// TIA Portal V18 export
// export: Created 2026-01-09T11:31:59.1599662Z, ExportSetting WithDefaults, DisplayName Totally Integrated Automation Portal, DisplayVersion V18 Update 5, DisplayName TIA Portal Openness, DisplayVersion V18 Update 5, DisplayName TIA Portal Teamcenter Gateway, DisplayVersion V18, DisplayName TIA Portal Version Control Interface, DisplayVersion V18, DisplayName SINAMICS Startdrive Advanced, DisplayVersion V18 SP2 Update 1, DisplayName SINAMICS Startdrive G110M, G120, G120C, G120D, G120P, G115D, DisplayVersion V18 SP2 Update 1, DisplayName SINAMICS Startdrive G130, G150, S120, S150, SINAMICS MV, S210, G220, S200, DisplayVersion V18 SP2 Update 1, DisplayName STEP 7 Professional, DisplayVersion V18 Update 5, DisplayName STEP 7 Safety, DisplayVersion V18, DisplayName WinCC Professional, DisplayVersion V18 Update 5
TagTable "WarningWord"
  GlobalWarning_01 : Word  (%DB1068.DBW0, CPU S71500-2PN_TP700, 100 ms)
  GlobalWarning_02 : Word  (%DB1068.DBW2, CPU S71500-2PN_TP700, 100 ms)
  GlobalWarning_03 : Word  (%DB1068.DBW4, CPU S71500-2PN_TP700, 100 ms)
  GlobalWarning_04 : Word  (%DB1068.DBW6, CPU S71500-2PN_TP700, 100 ms)
  GlobalWarning_05 : Word  (%DB1068.DBW8, CPU S71500-2PN_TP700, 100 ms)
  GlobalWarning_06 : Word  (%DB1068.DBW10, CPU S71500-2PN_TP700, 100 ms)
  GlobalWarning_07 : Word  (%DB1068.DBW12, CPU S71500-2PN_TP700, 100 ms)
  GlobalWarning_08 : Word  (%DB1068.DBW14, CPU S71500-2PN_TP700, 100 ms)
  GlobalWarning_09 : Word  (%DB1068.DBW16, CPU S71500-2PN_TP700, 100 ms)
  GlobalWarning_10 : Word  (%DB1068.DBW18, CPU S71500-2PN_TP700, 100 ms)
  IndexTableWarning_01 : Word  (%DB1068.DBW20, CPU S71500-2PN_TP700, 100 ms)
  IndexTableWarning_02 : Word  (%DB1068.DBW22, CPU S71500-2PN_TP700, 100 ms)
  ServoWarning_01 : Word  (%DB1068.DBW24, CPU S71500-2PN_TP700, 100 ms)
  ServoWarning_02 : Word  (%DB1068.DBW26, CPU S71500-2PN_TP700, 100 ms)
  ServePressWarning_01 : Word  (%DB1068.DBW28, CPU S71500-2PN_TP700, 100 ms)
  ServePressWarning_02 : Word  (%DB1068.DBW30, CPU S71500-2PN_TP700, 100 ms)
  3AxisInterpolationWarning_01 : Word  (%DB1068.DBW32, CPU S71500-2PN_TP700, 100 ms)
  3AxisInterpolationWarning_02 : Word  (%DB1068.DBW34, CPU S71500-2PN_TP700, 100 ms)
  LaserWeldingWarning_01 : Word  (%DB1068.DBW36, CPU S71500-2PN_TP700, 100 ms)
  LaserWeldingWarning_02 : Word  (%DB1068.DBW38, CPU S71500-2PN_TP700, 100 ms)
  LaserMarkingWarning_01 : Word  (%DB1068.DBW40, CPU S71500-2PN_TP700, 100 ms)
  LaserMarkingWarning_02 : Word  (%DB1068.DBW42, CPU S71500-2PN_TP700, 100 ms)
  PrinterWarning_01 : Word  (%DB1068.DBW44, CPU S71500-2PN_TP700, 100 ms)
  PrinterWarning_02 : Word  (%DB1068.DBW46, CPU S71500-2PN_TP700, 100 ms)
  MarkingWarning_01 : Word  (%DB1068.DBW48, CPU S71500-2PN_TP700, 100 ms)
  MarkingWarning_02 : Word  (%DB1068.DBW50, CPU S71500-2PN_TP700, 100 ms)
  LabellingWarning_01 : Word  (%DB1068.DBW52, CPU S71500-2PN_TP700, 100 ms)
  LabellingWarning_02 : Word  (%DB1068.DBW54, CPU S71500-2PN_TP700, 100 ms)
  DispensingWarning_01 : Word  (%DB1068.DBW56, CPU S71500-2PN_TP700, 100 ms)
  DispensingWarning_02 : Word  (%DB1068.DBW58, CPU S71500-2PN_TP700, 100 ms)
  GreasingWarning_01 : Word  (%DB1068.DBW60, CPU S71500-2PN_TP700, 100 ms)
  GreasingWarning_02 : Word  (%DB1068.DBW62, CPU S71500-2PN_TP700, 100 ms)
  HotWindSystemWarning_01 : Word  (%DB1068.DBW64, CPU S71500-2PN_TP700, 100 ms)
  HotWindSystemWarning_02 : Word  (%DB1068.DBW66, CPU S71500-2PN_TP700, 100 ms)
  HighFrequencyHeatingWarning_01 : Word  (%DB1068.DBW68, CPU S71500-2PN_TP700, 100 ms)
  HighFrequencyHeatingWarning_02 : Word  (%DB1068.DBW70, CPU S71500-2PN_TP700, 100 ms)
  DegaussingWarning_01 : Word  (%DB1068.DBW72, CPU S71500-2PN_TP700, 100 ms)
  DegaussingWarning_02 : Word  (%DB1068.DBW74, CPU S71500-2PN_TP700, 100 ms)
  BowlFeederWarning_01 : Word  (%DB1068.DBW76, CPU S71500-2PN_TP700, 100 ms)
  BowlFeederWarning_02 : Word  (%DB1068.DBW78, CPU S71500-2PN_TP700, 100 ms)
  RiveterWarning_01 : Word  (%DB1068.DBW80, CPU S71500-2PN_TP700, 100 ms)
  RiveterWarning_02 : Word  (%DB1068.DBW82, CPU S71500-2PN_TP700, 100 ms)
  HydraulicSystemWarning_01 : Word  (%DB1068.DBW84, CPU S71500-2PN_TP700, 100 ms)
  HydraulicSystemWarning_02 : Word  (%DB1068.DBW86, CPU S71500-2PN_TP700, 100 ms)
  RobotWarning_01 : Word  (%DB1068.DBW88, CPU S71500-2PN_TP700, 100 ms)
  RobotWarning_02 : Word  (%DB1068.DBW90, CPU S71500-2PN_TP700, 100 ms)
  CameraWarning_01 : Word  (%DB1068.DBW92, CPU S71500-2PN_TP700, 100 ms)
  CameraWarning_02 : Word  (%DB1068.DBW94, CPU S71500-2PN_TP700, 100 ms)
  ScannnerWarning_01 : Word  (%DB1068.DBW96, CPU S71500-2PN_TP700, 100 ms)
  ScannnerWarning_02 : Word  (%DB1068.DBW98, CPU S71500-2PN_TP700, 100 ms)
  MeasureSensorWarning_01 : Word  (%DB1068.DBW100, CPU S71500-2PN_TP700, 100 ms)
  MeasureSensorWarning_02 : Word  (%DB1068.DBW102, CPU S71500-2PN_TP700, 100 ms)
  LeakageTesterWarning_01 : Word  (%DB1068.DBW104, CPU S71500-2PN_TP700, 100 ms)
  LeakageTesterWarning_02 : Word  (%DB1068.DBW106, CPU S71500-2PN_TP700, 100 ms)
  TestPowerWarning_01 : Word  (%DB1068.DBW108, CPU S71500-2PN_TP700, 100 ms)
  TestPowerWarning_02 : Word  (%DB1068.DBW110, CPU S71500-2PN_TP700, 100 ms)
  HighVoltageTestWarning_01 : Word  (%DB1068.DBW112, CPU S71500-2PN_TP700, 100 ms)
  HighVoltageTestWarning_02 : Word  (%DB1068.DBW114, CPU S71500-2PN_TP700, 100 ms)
  EOLFinalInspectionWarning_01 : Word  (%DB1068.DBW116, CPU S71500-2PN_TP700, 100 ms)
  EOLFinalInspectionWarning_02 : Word  (%DB1068.DBW118, CPU S71500-2PN_TP700, 100 ms)
  ScrewWarning_01 : Word  (%DB1068.DBW120, CPU S71500-2PN_TP700, 100 ms)
  ScrewWarning_02 : Word  (%DB1068.DBW122, CPU S71500-2PN_TP700, 100 ms)
  3AxisScrewEncoderWarning_01 : Word  (%DB1068.DBW124, CPU S71500-2PN_TP700, 100 ms)
  3AxisScrewEncoderWarning_02 : Word  (%DB1068.DBW126, CPU S71500-2PN_TP700, 100 ms)
  HeatingWarning_01 : Word  (%DB1068.DBW128, CPU S71500-2PN_TP700, 100 ms)
  HeatingWarning_02 : Word  (%DB1068.DBW130, CPU S71500-2PN_TP700, 100 ms)
  PressurizedOilAirCylinderWarning_01 : Word  (%DB1068.DBW132, CPU S71500-2PN_TP700, 100 ms)
  PressurizedOilAirCylinderWarning_02 : Word  (%DB1068.DBW134, CPU S71500-2PN_TP700, 100 ms)
  MobyWarning_01 : Word  (%DB1068.DBW136, CPU S71500-2PN_TP700, 100 ms)
  MobyWarning_02 : Word  (%DB1068.DBW138, CPU S71500-2PN_TP700, 100 ms)
  IPC_Warning_01 : Word  (%DB1068.DBW140, CPU S71500-2PN_TP700, 100 ms)
  IPC_Warning_02 : Word  (%DB1068.DBW142, CPU S71500-2PN_TP700, 100 ms)
  ValveIslandWarning_01 : Word  (%DB1068.DBW144, CPU S71500-2PN_TP700, 100 ms)
  ValveIslandWarning_02 : Word  (%DB1068.DBW146, CPU S71500-2PN_TP700, 100 ms)
  RFIDWarning_01 : Word  (%DB1068.DBW148, CPU S71500-2PN_TP700, 100 ms)
  RFIDWarning_02 : Word  (%DB1068.DBW150, CPU S71500-2PN_TP700, 100 ms)
  RemoteI_O_Warning_01 : Word  (%DB1068.DBW152, CPU S71500-2PN_TP700, 100 ms)
  RemoteI_O_Warning_02 : Word  (%DB1068.DBW154, CPU S71500-2PN_TP700, 100 ms)
  DP_PN_SlaveStationWarning_01 : Word  (%DB1068.DBW156, CPU S71500-2PN_TP700, 100 ms)
  DP_PN_SlaveStationWarning_02 : Word  (%DB1068.DBW158, CPU S71500-2PN_TP700, 100 ms)
  MSCOMM_Warning_01 : Word  (%DB1068.DBW160, CPU S71500-2PN_TP700, 100 ms)
  MSCOMM_Warning_02 : Word  (%DB1068.DBW162, CPU S71500-2PN_TP700, 100 ms)
  FlowtesterWarning_01 : Word  (%DB1068.DBW164, CPU S71500-2PN_TP700, 100 ms)
  FlowtesterWarning_02 : Word  (%DB1068.DBW166, CPU S71500-2PN_TP700, 100 ms)
  CurrentsTesterWarning_01 : Word  (%DB1068.DBW168, CPU S71500-2PN_TP700, 100 ms)
  CurrentsTesterWarning_02 : Word  (%DB1068.DBW170, CPU S71500-2PN_TP700, 100 ms)
  VoltageTesterWarning_01 : Word  (%DB1068.DBW172, CPU S71500-2PN_TP700, 100 ms)
  VoltageTesterWarning_02 : Word  (%DB1068.DBW174, CPU S71500-2PN_TP700, 100 ms)
  InductanceTesterWarning_01 : Word  (%DB1068.DBW176, CPU S71500-2PN_TP700, 100 ms)
  InductanceTesterWarning_02 : Word  (%DB1068.DBW178, CPU S71500-2PN_TP700, 100 ms)
  ResistanceTesterWarning_01 : Word  (%DB1068.DBW180, CPU S71500-2PN_TP700, 100 ms)
  ResistanceTesterWarning_02 : Word  (%DB1068.DBW182, CPU S71500-2PN_TP700, 100 ms)
  LCR_TesterWarning_01 : Word  (%DB1068.DBW184, CPU S71500-2PN_TP700, 100 ms)
  LCR_TesterWarning_02 : Word  (%DB1068.DBW186, CPU S71500-2PN_TP700, 100 ms)
  PressureDisplacementMonitorWarning_01 : Word  (%DB1068.DBW188, CPU S71500-2PN_TP700, 100 ms)
  PressureDisplacementMonitorWarning_02 : Word  (%DB1068.DBW190, CPU S71500-2PN_TP700, 100 ms)
  UltrasonicWeldingWarning_01 : Word  (%DB1068.DBW192, CPU S71500-2PN_TP700, 100 ms)
  UltrasonicWeldingWarning_02 : Word  (%DB1068.DBW194, CPU S71500-2PN_TP700, 100 ms)
  ElectricResistanceWeldingWarning_01 : Word  (%DB1068.DBW196, CPU S71500-2PN_TP700, 100 ms)
  ElectricResistanceWeldingWarning_02 : Word  (%DB1068.DBW198, CPU S71500-2PN_TP700, 100 ms)
